FUNCTION_BLOCK MotorControl
VAR_INPUT
	switchFor: BOOL;
	switchBack: BOOL;
	
END_VAR
VAR_OUTPUT
END_VAR
VAR
	switchActive: BOOL;
	countValue: WORD;
	
	CounterMotor: CTUD;
	TOF_0: TOF;
	TOF_1: TOF;
	TOF_2: TOF;
	TOF_3: TOF;
	TOF_4: TOF;
	TOF_5: TOF;
	TOF_6: TOF;
	TON_0: TON;
END_VAR

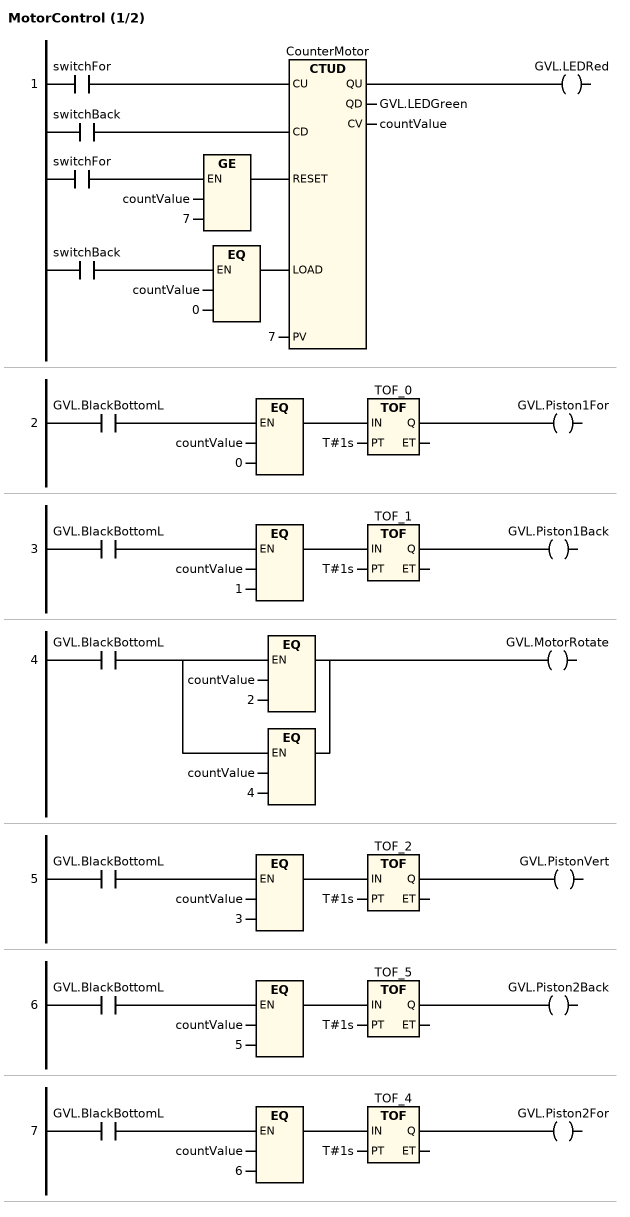
// NETWORK 1
CounterMotor(
    CU := switchFor,
    CD := switchBack,
    RESET := switchFor AND countValue >= 7,
    LOAD := switchBack AND countValue = 0,
    PV := 7,
    QD => GVL.LEDGreen,
    CV => countValue); // CTUD
GVL.LEDRed := CounterMotor.QU;

// NETWORK 2
TOF_0(IN := GVL.BlackBottomL AND countValue = 0, PT := T#1s); // TOF
GVL.Piston1For := TOF_0.Q;

// NETWORK 3
TOF_1(IN := GVL.BlackBottomL AND countValue = 1, PT := T#1s); // TOF
GVL.Piston1Back := TOF_1.Q;

// NETWORK 4
GVL.MotorRotate := GVL.BlackBottomL AND countValue = 2 OR GVL.BlackBottomL AND countValue = 4;

// NETWORK 5
TOF_2(IN := GVL.BlackBottomL AND countValue = 3, PT := T#1s); // TOF
GVL.PistonVert := TOF_2.Q;

// NETWORK 6
TOF_5(IN := GVL.BlackBottomL AND countValue = 5, PT := T#1s); // TOF
GVL.Piston2Back := TOF_5.Q;

// NETWORK 7
TOF_4(IN := GVL.BlackBottomL AND countValue = 6, PT := T#1s); // TOF
GVL.Piston2For := TOF_4.Q;

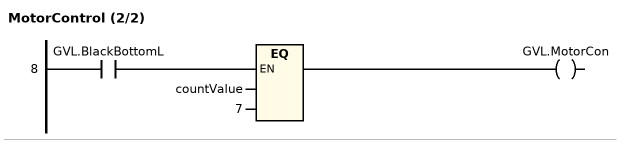
// NETWORK 8
GVL.MotorCon := GVL.BlackBottomL AND countValue = 7;

END_FUNCTION_BLOCK

(* stored: Version 1.1.0.1, ProductVersion 3.1.4024.12
   POU MotorControl: Id {bded6657-271f-4b86-b17e-96b11021a7c0}, SpecialFunc None *)
